TYPE ST_System_Bel_Zustand :
STRUCT
	Betrieb_Anford			: BOOL;
	Betrieb_Soll			: BOOL;
	Betrieb					: BOOL;
	Regelung_Modus			: SINT;
	Regelung_Sollw			: REAL;
	Regelung_Modus_Anford	: BOOL;

	Freigabe				: BOOL;
	Freigabe_Deakt			: BOOL;
	Freigabe_Code			: WORD;
	Stoerung				: BOOL;
	Stoerung_Code			: WORD;

	Warnung					: BOOL;
	Warnung_Code			: WORD;

	Farbcode			: STRING;

	Status					: SINT;
	Status_Vorl				: BOOL;
	Status_Nachl			: BOOL;

	Quittierung				: BOOL;

	Leistung				: REAL;

END_STRUCT
END_TYPE

(* stored: Version 1.1.0.1, ProductVersion 3.1.4024.10
   DUT ST_System_Bel_Zustand: Id {91444eb5-0729-4148-824f-b91bd91601e8} *)
